TYPE Sh10pilShutterConfig EXTENDS DeviceConfiguration :
STRUCT	
END_STRUCT
END_TYPE

(* stored: Version 1.1.0.1, ProductVersion 3.1.4024.4
   DUT Sh10pilShutterConfig: Id {c1127033-7121-46b1-b66e-56bfdcb2d87e} *)
